FUNCTION_BLOCK FB_ControlRampGenerator
VAR_INPUT
	input : RampGeneratorInput;
END_VAR
VAR
	state : E_RampGeneratorState := E_RampGeneratorState.End;
	rampGenerator : FB_CTRL_RAMP_GENERATOR;
	rampGeneratorParams	: ST_CTRL_RAMP_GENERATOR_PARAMS := (tTaskCycleTime := T#100MS, tCtrlCycleTime := T#100MS, fVeloPos := 0, fVeloNeg := 0);
END_VAR
VAR_OUTPUT
	rControlValue	: LREAL := 0;
	targetValueReached : BOOL := FALSE;
	isError : BOOL;
	eErrorID : E_CTRL_ERRORCODES;
END_VAR

IF input.restart = TRUE AND 0 <= input.rampTime AND rControlValue <> input.targetValue THEN
	state := E_RampGeneratorState.Init;
	input.restart := FALSE;
END_IF
	
CASE state OF
	E_RampGeneratorState.Init:
		IF 0 < input.rampTime THEN
			rampGeneratorParams.fVeloPos			:= ABS(input.targetValue - rControlValue) / input.rampTime * 0.1; (* in units per second *)
			rampGeneratorParams.fVeloNeg			:= rampGeneratorParams.fVeloPos; (* in units per second *)
			rampGenerator(bEnable := TRUE, fStart := rControlValue, fTarget:= input.targetValue, fOut => rControlValue, bValueReached => targetValueReached, bError => isError, eErrorID => eErrorID, stParams := rampGeneratorParams);
		ELSIF input.rampTime = 0 THEN
			rampGenerator(bEnable := FALSE, stParams := rampGeneratorParams);
			rampGeneratorParams.fVeloPos			:= input.targetValue; (* in units per second *)
			rampGeneratorParams.fVeloNeg			:= rampGeneratorParams.fVeloPos; (* in units per second *)
			rampGenerator(bEnable := TRUE, fStart := input.targetValue, fTarget:= input.targetValue, fOut => rControlValue, bValueReached => targetValueReached, bError => isError, eErrorID => eErrorID, stParams := rampGeneratorParams);
		END_IF
		state := E_RampGeneratorState.Run;
	
	E_RampGeneratorState.Run:
		rampGenerator(bEnable := TRUE, stParams := rampGeneratorParams, fOut => rControlValue, bValueReached => targetValueReached, bError => isError, eErrorID => eErrorID, stParams := rampGeneratorParams);
		IF targetValueReached = TRUE THEN
			state := E_RampGeneratorState.End;
		END_IF
		
	E_RampGeneratorState.End:
		rampGenerator(bEnable := FALSE, stParams := rampGeneratorParams, fOut => rControlValue);
END_CASE

END_FUNCTION_BLOCK

(* stored: Version 1.1.0.1, ProductVersion 3.1.4026.12
   POU FB_ControlRampGenerator: Id {a35b422b-580f-4aa7-bd81-602c2a7800da}, SpecialFunc None *)
